Fanuc TP program (LS listing): ZERO.LS

/PROG  ZERO
/ATTR
OWNER		= MNEDITOR;
COMMENT		= "";
PROG_SIZE	= 507;
CREATE		= DATE 23-10-17  TIME 10:32:56;
MODIFIED	= DATE 23-10-17  TIME 10:53:50;
FILE_NAME	= ;
VERSION		= 0;
LINE_COUNT	= 1;
MEMORY_SIZE	= 875;
PROTECT		= READ_WRITE;
TCD:  STACK_SIZE	= 0,
      TASK_PRIORITY	= 50,
      TIME_SLICE	= 0,
      BUSY_LAMP_OFF	= 0,
      ABORT_REQUEST	= 0,
      PAUSE_REQUEST	= 0;
DEFAULT_GROUP	= 1,*,*,*,*;
CONTROL_CODE	= 00000000 00000000;
LOCAL_REGISTERS	= 0,0,0;
/APPL
/APPL

AUTO_SINGULARITY_HEADER;
  ENABLE_SINGULARITY_AVOIDANCE   : FALSE;

PLTZ_MODE_HEADER;
 PLTZ_MODE_ENABLE   : FALSE;
 J4TURN  : ZERORAD;
 ORIENT  : DOWNWARDS;
/MN
   1:J P[1] 100% CNT100    ;
/POS
P[1]{
   GP1:
	UF : 0, UT : 1,
	J1=     0.000000 deg,	J2=     0.000000 deg,	J3=     0.000000 deg,
	J4=     0.000000 deg,	J5=   -90.000000 deg,	J6=   -90.000000 deg
};
/END
